// TwinCAT 3 PLC project PLC_A0
// ProgramVersion: 3.1.4024.0
// libraries:
//   Tc2_Standard, * (Beckhoff Automation GmbH)
//   Tc2_System, * (Beckhoff Automation GmbH)
//   Tc3_Module, * (Beckhoff Automation GmbH)
//   VisuSymbols,3.5.10.0,System
// project tree:
//   DT/ motorDUT.TcDUT
//   FB/ motorFB.TcPOU
//   / GlobalTextList.TcGTLO, PlcTask.TcTTO, Visualization Manager.TcVMO (not stored)
//   GVLs/ GVL.TcGVL, IO.TcGVL
//   POUs/ automat_PRG.TcPOU, motor_PRG.TcPOU, PLC_PRG.TcPOU
//   VISUs/ Visualization.TcVIS
// real-time tasks:
//   TASK PlcTask: cycle T#10ms, priority 6, ADS port 350
// I/O:
//   DEVICE master EtherCaT, AmsNetId 192.168.0.237.3.1
//     A1 [EP1008-0001 8 Ch. Dig. Input 24V, 3ms, M8]
//     A2 [EP2001-1000 8 Ch. Dig. Output 24V, 0,5A, M8]
// variable links:
//   PLC_A0/PLC_A0 Instance <-> master EtherCaT/A1
//     PlcTask Inputs/IO.A1_DI{0..7} <-> Channel {1..8}/A1_DI{0..7}  (8 links)
//   PLC_A0/PLC_A0 Instance <-> master EtherCaT/A2
//     PlcTask Outputs/IO.A2_DO0 <-> Group 0/A2_DO0
//     PlcTask Outputs/IO.A2_DO1 <-> Group 0/A2_DO1
//     PlcTask Outputs/IO.A2_DO2 <-> Group 0/A2_DO2
//     PlcTask Outputs/IO.A2_DO3 <-> Group 0/A2_DO3
//     PlcTask Outputs/IO.A2_DO4 <-> Group 1/A2_DO4
//     PlcTask Outputs/IO.A2_DO5 <-> Group 1/A2_DO5
//     PlcTask Outputs/IO.A2_DO6 <-> Group 1/A2_DO6
//     PlcTask Outputs/IO.A2_DO7 <-> Group 1/A2_DO7

CONFIGURATION PLC_A0
    RESOURCE PLC ON TwinCAT3
        TASK PlcTask(INTERVAL := T#10ms, PRIORITY := 6);
        PROGRAM PLC_PRG WITH PlcTask : PLC_PRG;
        PROGRAM motor_PRG WITH PlcTask : motor_PRG;
    END_RESOURCE
END_CONFIGURATION

// ---- DT/motorDUT.TcDUT
TYPE motorDUT :
STRUCT
	en: BOOL; //start/stop motor	

	Amax: REAL; //maximal acceleration
	VMax: REAL; //maximal velocity 
	VAct: REAL; //actual velocity
	VSet: REAL; //requsted velocity
	
	dir:  BOOL; //actual direction
 
	SAct: REAL; //actual position
	SSet: real; //requested position
	Sreset: BOOL; //reset positon
	
	endPoint1 :BOOL;
	endPoint2 :BOOL;
END_STRUCT
END_TYPE

// ---- GVLs/GVL.TcGVL
{attribute 'qualified_only'}
VAR_GLOBAL
//motor global 
	motor1: motorDUT; 
	motor2: motorDUT;
// GUI
	StartStop: bool; //start and stop process  
END_VAR

// ---- GVLs/IO.TcGVL
{attribute 'qualified_only'}
VAR_GLOBAL
//inputs 
	A1_DI0 AT %I* : BOOL;	// safety
	A1_DI1 AT %I* : BOOL;	// cylinder sensor
	A1_DI2 AT %I* : BOOL;	// 1. Endpoint senzor - M1
	A1_DI3 AT %I* : BOOL;	// 2. Endpoint senzor - M1
	A1_DI4 AT %I* : BOOL;
	A1_DI5 AT %I* : BOOL;
	A1_DI6 AT %I* : BOOL;
	A1_DI7 AT %I* : BOOL;

	//output
	A2_DO0 AT %Q* : BOOL;	// start motor 1
	A2_DO1 AT %Q* : BOOL;	// direction motor 1
	A2_DO2 AT %Q* : BOOL;	// start motor 2
	A2_DO3 AT %Q* : BOOL;	//gripper finger
	A2_DO4 AT %Q* : BOOL;
	A2_DO5 AT %Q* : BOOL;
	A2_DO6 AT %Q* : BOOL;
	A2_DO7 AT %Q* : BOOL;
END_VAR

// ---- POUs/PLC_PRG.TcPOU
PROGRAM PLC_PRG
VAR
//triggers
	trigA0_DI1: R_TRIG;	//trigger for cylinder sensor 

	trigStart: R_TRIG;
END_VAR

// triggers
trigA0_DI1(clk := IO.A1_DI1);
trigStart (clk := gvl.StartStop); 


//calling program 
automat_PRG(SFCInit := trigStart.Q);

END_PROGRAM

// ---- POUs/automat_PRG.TcPOU
PROGRAM automat_PRG
VAR_INPUT
SFCInit: BOOL; 
END_VAR
VAR
	counter: INT; //counting cyklus
END_VAR

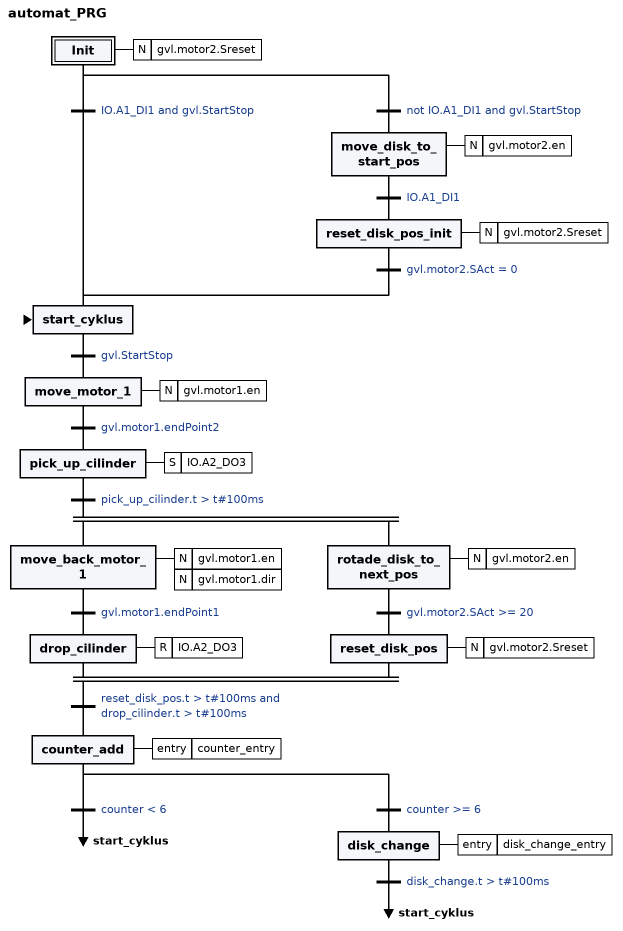
INITIAL_STEP Init:
    gvl.motor2.Sreset(N);
END_STEP
TRANSITION FROM Init TO start_cyklus
    := IO.A1_DI1 and gvl.StartStop;
END_TRANSITION
TRANSITION FROM Init TO move_disk_to_start_pos
    := not IO.A1_DI1 and gvl.StartStop;
END_TRANSITION
STEP move_disk_to_start_pos:
    gvl.motor2.en(N);
END_STEP
TRANSITION FROM move_disk_to_start_pos TO reset_disk_pos_init
    := IO.A1_DI1;
END_TRANSITION
STEP reset_disk_pos_init:
    gvl.motor2.Sreset(N);
END_STEP
TRANSITION FROM reset_disk_pos_init TO start_cyklus
    := gvl.motor2.SAct = 0;
END_TRANSITION
STEP start_cyklus:
END_STEP
TRANSITION FROM start_cyklus TO move_motor_1
    := gvl.StartStop;
END_TRANSITION
STEP move_motor_1:
    gvl.motor1.en(N);
END_STEP
TRANSITION FROM move_motor_1 TO pick_up_cilinder
    := gvl.motor1.endPoint2;
END_TRANSITION
STEP pick_up_cilinder:
    IO.A2_DO3(S);
END_STEP
TRANSITION FROM pick_up_cilinder TO (move_back_motor_1, rotade_disk_to_next_pos)
    := pick_up_cilinder.t > t#100ms;
END_TRANSITION
STEP move_back_motor_1:
    gvl.motor1.en(N);
    gvl.motor1.dir(N);
END_STEP
TRANSITION FROM move_back_motor_1 TO drop_cilinder
    := gvl.motor1.endPoint1;
END_TRANSITION
STEP drop_cilinder:
    IO.A2_DO3(R);
END_STEP
STEP rotade_disk_to_next_pos:
    gvl.motor2.en(N);
END_STEP
TRANSITION FROM rotade_disk_to_next_pos TO reset_disk_pos
    := gvl.motor2.SAct >= 20;
END_TRANSITION
STEP reset_disk_pos:
    gvl.motor2.Sreset(N);
END_STEP
TRANSITION FROM (drop_cilinder, reset_disk_pos) TO counter_add
    := reset_disk_pos.t > t#100ms and drop_cilinder.t > t#100ms;
END_TRANSITION
STEP counter_add:
    counter_entry(P1);  // entry action
END_STEP
TRANSITION FROM counter_add TO start_cyklus
    := counter < 6;
END_TRANSITION
TRANSITION FROM counter_add TO disk_change
    := counter >= 6;
END_TRANSITION
STEP disk_change:
    disk_change_entry(P1);  // entry action
END_STEP
TRANSITION FROM disk_change TO start_cyklus
    := disk_change.t > t#100ms;
END_TRANSITION

ACTION counter_entry:
counter := counter + 1;
END_ACTION

ACTION disk_change_entry:
counter := 0;
END_ACTION

END_PROGRAM

// ---- POUs/motor_PRG.TcPOU
PROGRAM motor_PRG
VAR
	motor1_fb :motorFB;
	motor2_FB: motorFB;
END_VAR

// note: this text did not pass the execution check against the stored diagram
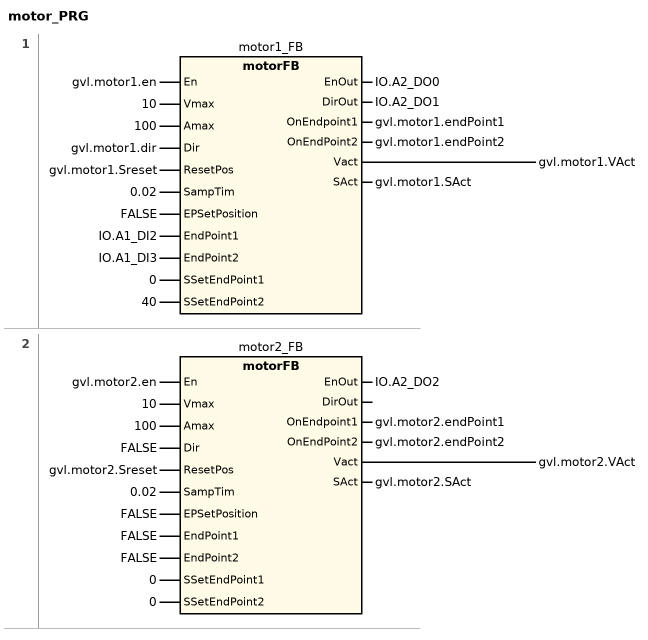
// NETWORK 1
motor1_FB(
    En := gvl.motor1.en,
    Vmax := 10,
    Amax := 100,
    Dir := gvl.motor1.dir,
    ResetPos := gvl.motor1.Sreset,
    SampTim := 0.02,
    EPSetPosition := FALSE,
    EndPoint1 := IO.A1_DI2,
    EndPoint2 := IO.A1_DI3,
    SSetEndPoint1 := 0,
    SSetEndPoint2 := 40,
    EnOut => IO.A2_DO0,
    DirOut => IO.A2_DO1,
    OnEndpoint1 => gvl.motor1.endPoint1,
    OnEndPoint2 => gvl.motor1.endPoint2,
    SAct => gvl.motor1.SAct); // motorFB
gvl.motor1.VAct := motor1_FB.Vact;

// NETWORK 2
motor2_FB(
    En := gvl.motor2.en,
    Vmax := 10,
    Amax := 100,
    Dir := FALSE,
    ResetPos := gvl.motor2.Sreset,
    SampTim := 0.02,
    EPSetPosition := FALSE,
    EndPoint1 := FALSE,
    EndPoint2 := FALSE,
    SSetEndPoint1 := 0,
    SSetEndPoint2 := 0,
    EnOut => IO.A2_DO2,
    OnEndpoint1 => gvl.motor2.endPoint1,
    OnEndPoint2 => gvl.motor2.endPoint2,
    SAct => gvl.motor2.SAct); // motorFB
gvl.motor2.VAct := motor2_FB.Vact;

END_PROGRAM

// ---- FB/motorFB.TcPOU
FUNCTION_BLOCK motorFB
VAR_INPUT
	En: BOOL; //motor start/stop 
	Vmax: REAL; //max velocity (un/sec)
	Amax: REAL; //max acceleration (un/sec^2)
	Dir: BOOL; //actual direction
	ResetPos: BOOL; //reseting position
	SampTim: REAL; //program cycle length (s) ¨
	EPSetPosition: BOOL; //if true and one of setpoint switch is pressed, set the position of endpoint switch
	EndPoint1 :BOOL;	//endpoint switch
	EndPoint2 :BOOL;	//endpoint switch
	SSetEndPoint1 :INT;		//set position on endpoint 1
	SSetEndPoint2 :INT; 	//set position on endPoint 2
END_VAR
VAR_OUTPUT
	EnOut: BOOL; //en output for DO
	DirOut: BOOL; //dir output for DO
	
	OnEndpoint1: BOOL; //EP switch is pressed
	OnEndPoint2: BOOL; //EP switch is pressed 
	
	Vact: REAL; //actual velocity(un/sec) 
	SAct: REAL; // actual position(un) 
END_VAR
VAR
	Vset: REAL; // internal variable for reqzest velocity 
	
	trigStart: R_TRIG; //trigger for starting process 
	trigResetPos: R_TRig; //trigger for reseting position
END_VAR

trigStart(clk := en); //start trigger
trigResetPos (clk := resetPos);

IF trigStart.Q THEN 
	Vset := Vmax; //count internal value for set velocity 
END_IF	

if en then 
	//counting act velocity
	IF Vset > Vact THEN //accelararion
		Vact := Vact + (Amax * sampTim);
	ELSIF Vset < Vact THEN //deceleration
		Vact := Vact - (Amax * sampTim);
	ELSE // on set speed (not needed, just for better understanding)
		Vact := Vset;
	END_IF
	
	//couning actual position
	IF NOT dir THEN
		SAct := SAct + (Vact*SampTim);
	ELSE
		SAct := SAct - (Vact*SampTim);
	END_IF	
//if the motor is turned off, it resets the variables
ELSE
	//velocity  
	Vact := 0;
	Vset := 0;
	//position reset 
	IF trigResetPos.Q THEN
		Sact := 0;
	END_IF
END_IF

//endpoint switches
IF EPSetPosition THEN
	IF EndPoint1 THEN 
		Sact := SSetEndPoint1;
	ELSIF Endpoint2 THEN
		Sact := SSetEndPoint2;
	END_IF
END_IF

//output
OnEndpoint1 := EndPoint1; 
OnEndpoint2 := EndPoint2; 

enOut := en; 
dirOut := dir;

END_FUNCTION_BLOCK

// ---- GlobalTextList.TcGTLO
TEXTLIST GlobalTextList
  708 = '%2.1f'
  437 = 'Counter:'
  302 = 'cylinder sensor'
  253 = 'EndPoint 1'
  705 = 'EndPoint 2'
  170 = 'Grapper: '
  735 = 'Motor 1'
  626 = 'Motor 2'
  881 = 'SAct:'
  900 = 'start'
  517 = 'VAct:'
END_TEXTLIST

// ---- VISUs/Visualization.TcVIS
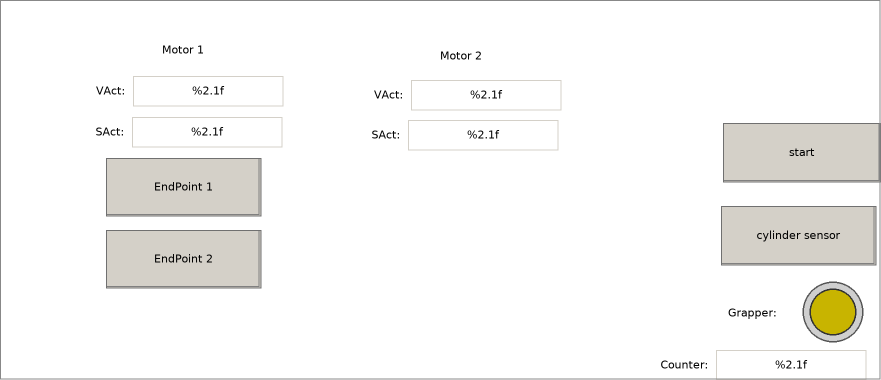
VISUALIZATION Visualization  // 881x380
    Button (723,123 158x59), "start"
        toggle GVL.StartStop
    Button (721,206 155x59), "cylinder sensor"
        toggle IO.A1_DI1
    Button (106,158 155x58), "EndPoint 1"
        tap IO.A1_DI2
    Button (106,230 155x58), "EndPoint 2"
        tap IO.A1_DI3
    Label (108,35 150x30), "Motor 1"
    Group (83,76 200x30)
        Label (0,0 45x30), "VAct:"
        Textfield (50,0 150x30), "%2.1f", text variable: GVL.motor1.VAct
    Group (84,117 198x30)
        Label (0,0 43x30), "SAct:"
        Textfield (48,0 150x30), "%2.1f", text variable: GVL.motor1.SAct
    Label (386,41 150x30), "Motor 2"
    Group (362,80 199x30)
        Label (0,0 44x30), "VAct:"
        Textfield (49,0 150x30), "%2.1f", text variable: GVL.motor2.VAct
    Group (365,120 193x30)
        Label (0,0 38x30), "SAct:"
        Textfield (43,0 150x30), "%2.1f", text variable: GVL.motor2.SAct
    Label (679,298 150x30), "Grapper:"
    Lamp1 (798,277 70x70), variable: A0_DO3, style: Lamp-Lamp1-Yellow
    Label (583,350 128x30), "Counter:"
    Textfield (716,350 150x30), "%2.1f", text variable: automat_PRG.counter
END_VISUALIZATION
